(* IEC 61131-3 sources: Proyecto_test/src, 4 files *)

(* ---- myfc.st ---- *)
FUNCTION myfc: INT
    VAR_INPUT

    END_VAR
    ;
END_FUNCTION

FUNCTION_BLOCK myfb
    VAR_INPUT
        myinput1: INT;
        myinput2: REAL;
        myinput3: INT;
    END_VAR

VAR
    myglobalstate: INT;
END_VAR

VAR_OUTPUT

    data: INT;

END_VAR

data := myinput1;

END_FUNCTION_BLOCK

TYPE
    mystruct : STRUCT
        Member1: INT;
        member2:INT;
        member3:INT;
    END_STRUCT;
END_TYPE

(* ---- configuration.st ---- *)
CONFIGURATION MyConfiguration
    TASK Main(Interval := T#1000ms, Priority := 1);
    TASK Background(PRIORITY:=1);
    PROGRAM P1 WITH Main: MyProgram;
    PROGRAM P2 WITH Background: MyProgram2;

    VAR_GLOBAL

        MyhardwareInput AT %I0.0: bool;
        MyhardwareOutput AT %QW4:INT;

    END_VAR

    VAR_GLOBAL

        Myglobalstorage : INT;
    END_VAR

    VAR_GLOBAL CONSTANT

        myglobalconstant : INT :=5;

    END_VAR

END_CONFIGURATION

(* ---- program copy.st ---- *)
PROGRAM MyProgram2
    VAR_EXTERNAL

    END_VAR

    VAR

    END_VAR

    VAR_TEMP

    END_VAR

    // code here
    ;
END_PROGRAM

(* ---- program.st ---- *)
PROGRAM MyProgram
    VAR_EXTERNAL

        Myglobalstorage : INT;
    END_VAR

    VAR

        myfbinstance:myfb;

    END_VAR

    VAR_TEMP

    END_VAR

    myfbinstance(3,5,6);
    myglobalstorage:= myfbinstance.data;

    // code here
    ;
END_PROGRAM
